Staubli VAL3: refreshDynamic.pgx

program refreshDynamic()
begin
  // DO NOT CHANGE
  nRefresh=clock()
  //
  // ADD HERE
  //
  call CycleRefresh()
  //
  use:bUseRefresh=false
end
